// TIA Portal V19 export
TYPE "UDT_SIM_REAL"
   STRUCT
      en : Bool;
      value : Real;
   END_STRUCT;
END_TYPE
